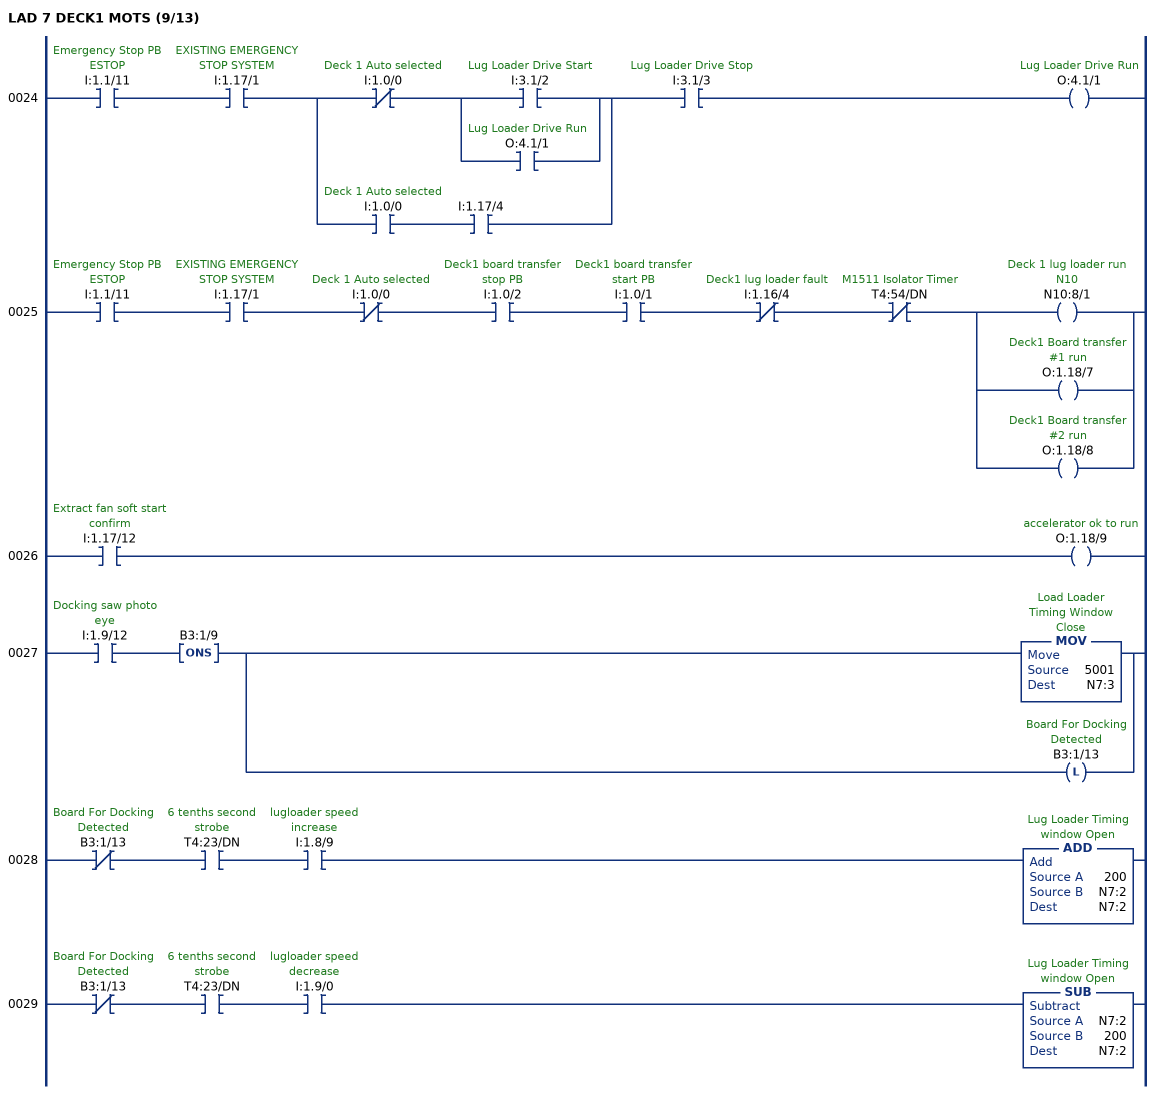
% Rung: 24 %
SOR XIC I:1.1/11 XIC I:1.17/1 BST XIO I:1.0/0 BST XIC I:3.1/2 NXB XIC O:4.1/1 BND NXB XIC I:1.0/0 XIC I:1.17/4 BND XIC I:3.1/3 OTE O:4.1/1 EOR
%   I:1.1/11  ESTOP  "Emergency Stop PB" %
%   I:1.17/1  "EXISTING EMERGENCY STOP SYSTEM" %
%   I:1.0/0  "Deck 1 Auto selected" %
%   I:3.1/2  "Lug Loader Drive Start" %
%   O:4.1/1  "Lug Loader Drive Run" %
%   I:3.1/3  "Lug Loader Drive Stop" %
% Rung: 25 %
SOR XIC I:1.1/11 XIC I:1.17/1 XIO I:1.0/0 XIC I:1.0/2 XIC I:1.0/1 XIO I:1.16/4 XIO T4:54/DN BST OTE N10:8/1 NXB OTE O:1.18/7 NXB OTE O:1.18/8 BND EOR
%   I:1.1/11  ESTOP  "Emergency Stop PB" %
%   I:1.17/1  "EXISTING EMERGENCY STOP SYSTEM" %
%   I:1.0/0  "Deck 1 Auto selected" %
%   I:1.0/2  "Deck1 board transfer stop PB" %
%   I:1.0/1  "Deck1 board transfer start PB" %
%   I:1.16/4  "Deck1 lug loader fault" %
%   T4:54  "M1511 Isolator Timer" %
%   N10:8/1  N10  "Deck 1 lug loader run" %
%   O:1.18/7  "Deck1 Board transfer #1 run" %
%   O:1.18/8  "Deck1 Board transfer #2 run" %
% Rung: 26 %
SOR XIC I:1.17/12 OTE O:1.18/9 EOR
%   I:1.17/12  "Extract fan soft start confirm" %
%   O:1.18/9  "accelerator ok to run" %
% Rung: 27 %
SOR XIC I:1.9/12 OSR B3:1/9 BST MOV 5001 N7:3 NXB OTL B3:1/13 BND EOR
%   I:1.9/12  "Docking saw photo eye" %
%   N7:3  "Load Loader Timing Window Close" %
%   B3:1/13  "Board For Docking Detected" %
% Rung: 28 %
SOR XIO B3:1/13 XIC T4:23/DN XIC I:1.8/9 ADD 200 N7:2 N7:2 EOR
%   B3:1/13  "Board For Docking Detected" %
%   T4:23/DN  "6 tenths second strobe" %
%   I:1.8/9  "lugloader speed increase" %
%   N7:2  "Lug Loader Timing window Open" %
% Rung: 29 %
SOR XIO B3:1/13 XIC T4:23/DN XIC I:1.9/0 SUB N7:2 200 N7:2 EOR
%   B3:1/13  "Board For Docking Detected" %
%   T4:23/DN  "6 tenths second strobe" %
%   I:1.9/0  "lugloader speed decrease" %
%   N7:2  "Lug Loader Timing window Open" %

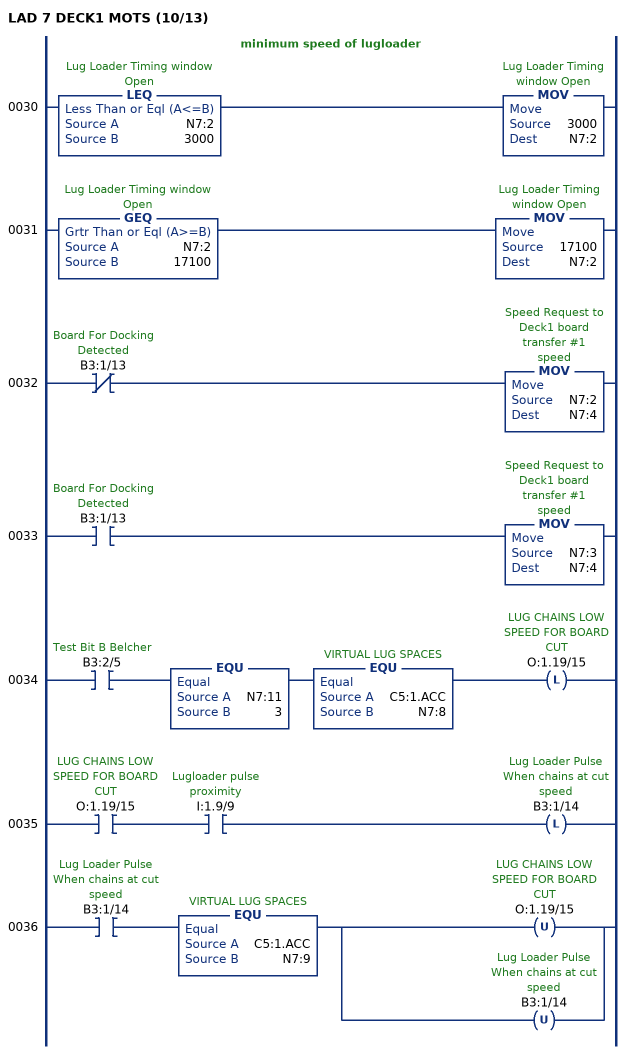
% Rung: 30 %
% TITLE: minimum speed of lugloader %
SOR LEQ N7:2 3000 MOV 3000 N7:2 EOR
%   N7:2  "Lug Loader Timing window Open" %
% Rung: 31 %
SOR GEQ N7:2 17100 MOV 17100 N7:2 EOR
%   N7:2  "Lug Loader Timing window Open" %
% Rung: 32 %
SOR XIO B3:1/13 MOV N7:2 N7:4 EOR
%   B3:1/13  "Board For Docking Detected" %
%   N7:2  "Lug Loader Timing window Open" %
%   N7:4  "Speed Request to Deck1 board transfer #1 speed" %
% Rung: 33 %
SOR XIC B3:1/13 MOV N7:3 N7:4 EOR
%   B3:1/13  "Board For Docking Detected" %
%   N7:3  "Load Loader Timing Window Close" %
%   N7:4  "Speed Request to Deck1 board transfer #1 speed" %
% Rung: 34 %
SOR XIC B3:2/5 EQU N7:11 3 EQU C5:1.ACC N7:8 OTL O:1.19/15 EOR
%   B3:2/5  "Test Bit B Belcher" %
%   C5:1  "VIRTUAL LUG SPACES" %
%   N7:8  "CUT BOARD SLOW DOWN ON" %
%   O:1.19/15  "LUG CHAINS LOW SPEED FOR BOARD CUT" %
% Rung: 35 %
SOR XIC O:1.19/15 XIC I:1.9/9 OTL B3:1/14 EOR
%   O:1.19/15  "LUG CHAINS LOW SPEED FOR BOARD CUT" %
%   I:1.9/9  "Lugloader pulse proximity" %
%   B3:1/14  "Lug Loader Pulse When chains at cut speed" %
% Rung: 36 %
SOR XIC B3:1/14 EQU C5:1.ACC N7:9 BST OTU O:1.19/15 NXB OTU B3:1/14 BND EOR
%   B3:1/14  "Lug Loader Pulse When chains at cut speed" %
%   C5:1  "VIRTUAL LUG SPACES" %
%   O:1.19/15  "LUG CHAINS LOW SPEED FOR BOARD CUT" %

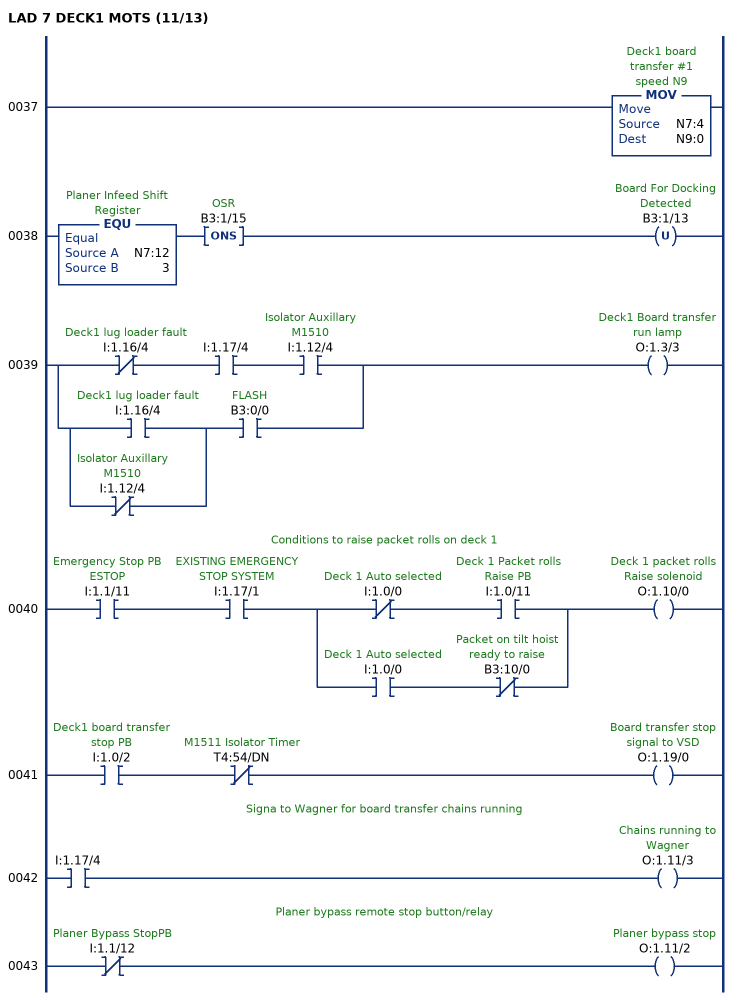
% Rung: 37 %
SOR MOV N7:4 N9:0 EOR
%   N7:4  "Speed Request to Deck1 board transfer #1 speed" %
%   N9:0  N9  "Deck1 board transfer #1 speed" %
% Rung: 38 %
SOR EQU N7:12 3 OSR B3:1/15 OTU B3:1/13 EOR
%   N7:12  "Planer Infeed Shift Register" %
%   B3:1/15  "OSR" %
%   B3:1/13  "Board For Docking Detected" %
% Rung: 39 %
SOR BST XIO I:1.16/4 XIC I:1.17/4 XIC I:1.12/4 NXB BST XIC I:1.16/4 NXB XIO I:1.12/4 BND XIC B3:0/0 BND OTE O:1.3/3 EOR
%   I:1.16/4  "Deck1 lug loader fault" %
%   I:1.12/4  "Isolator Auxillary M1510" %
%   B3:0/0  FLASH %
%   O:1.3/3  "Deck1 Board transfer run lamp" %
% Rung: 40 %
% Conditions to raise packet rolls on deck 1 %
SOR XIC I:1.1/11 XIC I:1.17/1 BST XIO I:1.0/0 XIC I:1.0/11 NXB XIC I:1.0/0 XIO B3:10/0 BND OTE O:1.10/0 EOR
%   I:1.1/11  ESTOP  "Emergency Stop PB" %
%   I:1.17/1  "EXISTING EMERGENCY STOP SYSTEM" %
%   I:1.0/0  "Deck 1 Auto selected" %
%   I:1.0/11  "Deck 1 Packet rolls Raise PB" %
%   B3:10/0  "Packet on tilt hoist ready to raise" %
%   O:1.10/0  "Deck 1 packet rolls Raise solenoid" %
% Rung: 41 %
SOR XIC I:1.0/2 XIO T4:54/DN OTE O:1.19/0 EOR
%   I:1.0/2  "Deck1 board transfer stop PB" %
%   T4:54  "M1511 Isolator Timer" %
%   O:1.19/0  "Board transfer stop signal to VSD" %
% Rung: 42 %
% Signa to Wagner for board transfer chains running %
SOR XIC I:1.17/4 OTE O:1.11/3 EOR
%   O:1.11/3  "Chains running to Wagner" %
% Rung: 43 %
% Planer bypass remote stop button/relay %
SOR XIO I:1.1/12 OTE O:1.11/2 EOR
%   I:1.1/12  "Planer Bypass StopPB" %
%   O:1.11/2  "Planer bypass stop" %

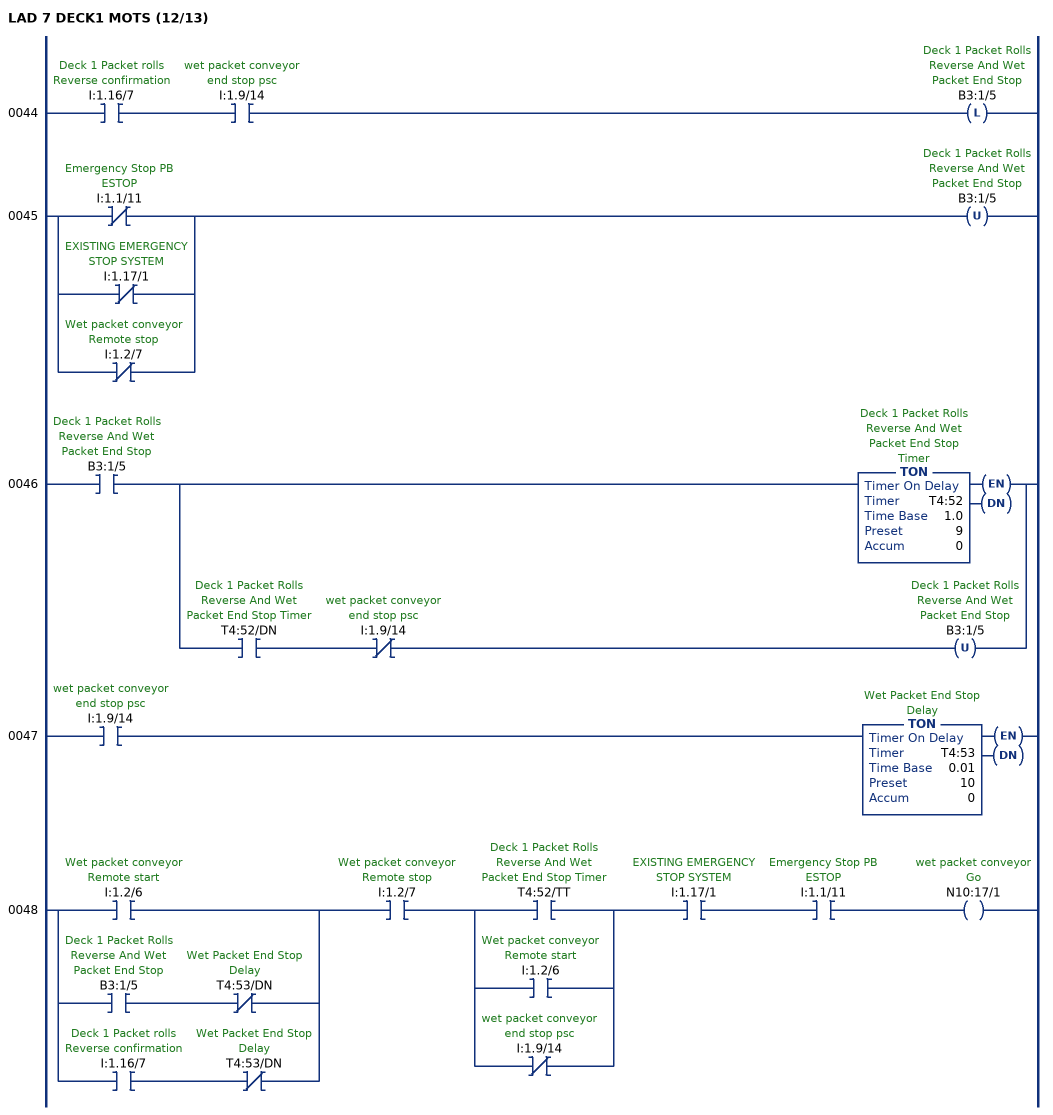
% Rung: 44 %
SOR XIC I:1.16/7 XIC I:1.9/14 OTL B3:1/5 EOR
%   I:1.16/7  "Deck 1 Packet rolls Reverse confirmation" %
%   I:1.9/14  "wet packet conveyor end stop psc" %
%   B3:1/5  "Deck 1 Packet Rolls Reverse And Wet Packet End Stop" %
% Rung: 45 %
SOR BST XIO I:1.1/11 NXB XIO I:1.17/1 NXB XIO I:1.2/7 BND OTU B3:1/5 EOR
%   I:1.1/11  ESTOP  "Emergency Stop PB" %
%   I:1.17/1  "EXISTING EMERGENCY STOP SYSTEM" %
%   I:1.2/7  "Wet packet conveyor Remote stop" %
%   B3:1/5  "Deck 1 Packet Rolls Reverse And Wet Packet End Stop" %
% Rung: 46 %
SOR XIC B3:1/5 BST TON T4:52 1.0 9 0 NXB XIC T4:52/DN XIO I:1.9/14 OTU B3:1/5 BND EOR
%   B3:1/5  "Deck 1 Packet Rolls Reverse And Wet Packet End Stop" %
%   T4:52  "Deck 1 Packet Rolls Reverse And Wet Packet End Stop Timer" %
%   I:1.9/14  "wet packet conveyor end stop psc" %
% Rung: 47 %
SOR XIC I:1.9/14 TON T4:53 0.01 10 0 EOR
%   I:1.9/14  "wet packet conveyor end stop psc" %
%   T4:53  "Wet Packet End Stop Delay" %
% Rung: 48 %
SOR BST XIC I:1.2/6 NXB XIC B3:1/5 XIO T4:53/DN NXB XIC I:1.16/7 XIO T4:53/DN BND XIC I:1.2/7 BST XIC T4:52/TT NXB XIC I:1.2/6 NXB XIO I:1.9/14 BND XIC I:1.17/1 XIC I:1.1/11 OTE N10:17/1 EOR
%   I:1.2/6  "Wet packet conveyor Remote start" %
%   B3:1/5  "Deck 1 Packet Rolls Reverse And Wet Packet End Stop" %
%   T4:53  "Wet Packet End Stop Delay" %
%   I:1.16/7  "Deck 1 Packet rolls Reverse confirmation" %
%   I:1.2/7  "Wet packet conveyor Remote stop" %
%   T4:52  "Deck 1 Packet Rolls Reverse And Wet Packet End Stop Timer" %
%   I:1.9/14  "wet packet conveyor end stop psc" %
%   I:1.17/1  "EXISTING EMERGENCY STOP SYSTEM" %
%   I:1.1/11  ESTOP  "Emergency Stop PB" %
%   N10:17/1  "wet packet conveyor Go" %

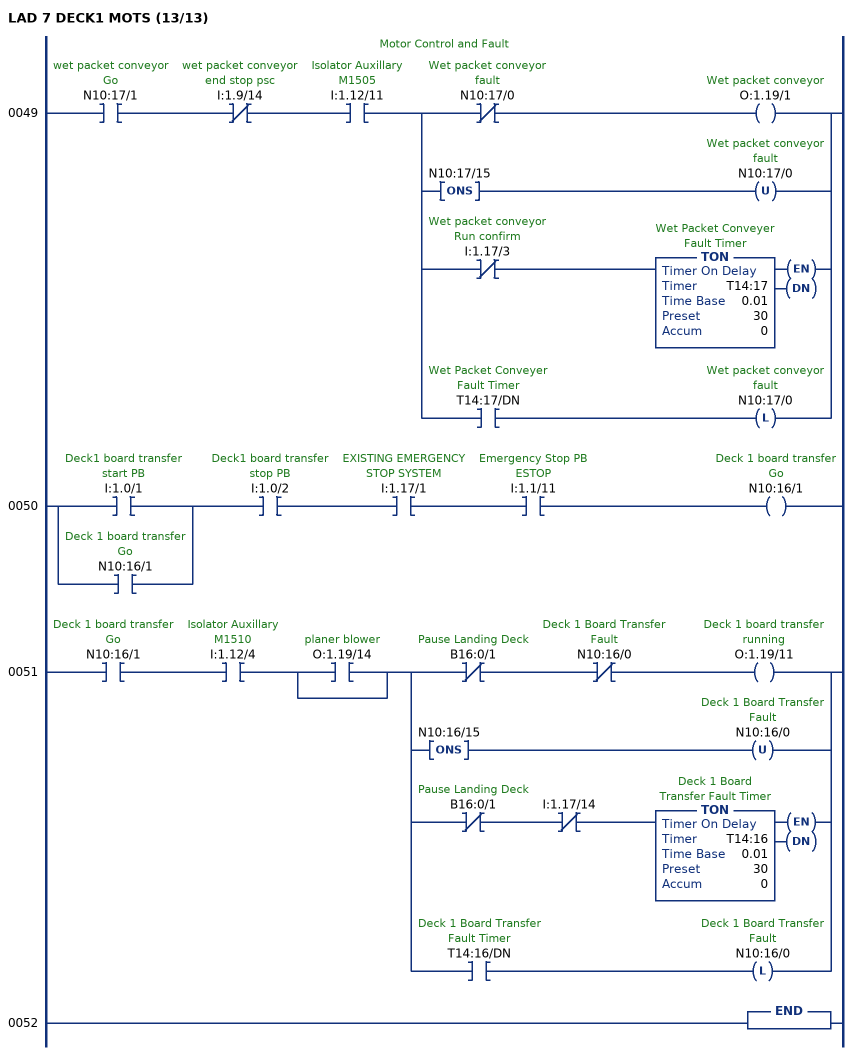
% Rung: 49 %
% Motor Control and Fault %
SOR XIC N10:17/1 XIO I:1.9/14 XIC I:1.12/11 BST XIO N10:17/0 OTE O:1.19/1 NXB OSR N10:17/15 OTU N10:17/0 NXB XIO I:1.17/3 TON T14:17 0.01 30 0 NXB XIC T14:17/DN OTL N10:17/0 BND EOR
%   N10:17/1  "wet packet conveyor Go" %
%   I:1.9/14  "wet packet conveyor end stop psc" %
%   I:1.12/11  "Isolator Auxillary M1505" %
%   N10:17/0  "Wet packet conveyor fault" %
%   O:1.19/1  "Wet packet conveyor" %
%   I:1.17/3  "Wet packet conveyor Run confirm" %
%   T14:17  "Wet Packet Conveyer Fault Timer" %
% Rung: 50 %
SOR BST XIC I:1.0/1 NXB XIC N10:16/1 BND XIC I:1.0/2 XIC I:1.17/1 XIC I:1.1/11 OTE N10:16/1 EOR
%   I:1.0/1  "Deck1 board transfer start PB" %
%   N10:16/1  "Deck 1 board transfer Go" %
%   I:1.0/2  "Deck1 board transfer stop PB" %
%   I:1.17/1  "EXISTING EMERGENCY STOP SYSTEM" %
%   I:1.1/11  ESTOP  "Emergency Stop PB" %
% Rung: 51 %
SOR XIC N10:16/1 XIC I:1.12/4 BST XIC O:1.19/14 NXB BND BST XIO B16:0/1 XIO N10:16/0 OTE O:1.19/11 NXB OSR N10:16/15 OTU N10:16/0 NXB XIO B16:0/1 XIO I:1.17/14 TON T14:16 0.01 30 0 NXB XIC T14:16/DN OTL N10:16/0 BND EOR
%   N10:16/1  "Deck 1 board transfer Go" %
%   I:1.12/4  "Isolator Auxillary M1510" %
%   O:1.19/14  "planer blower" %
%   B16:0/1  "Pause Landing Deck" %
%   N10:16/0  "Deck 1 Board Transfer Fault" %
%   O:1.19/11  "Deck 1 board transfer running" %
%   T14:16  "Deck 1 Board Transfer Fault Timer" %
% Rung: 52 %
SOR END EOR

LADDER 8 "EXTRACTFAN"
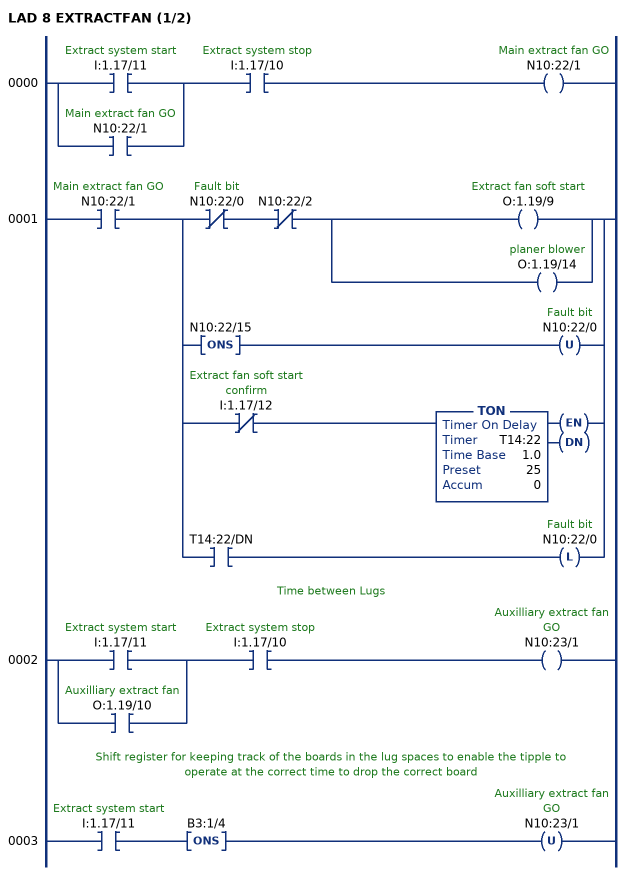
% Rung: 0 %
SOR BST XIC I:1.17/11 NXB XIC N10:22/1 BND XIC I:1.17/10 OTE N10:22/1 EOR
%   I:1.17/11  "Extract system start" %
%   N10:22/1  "Main extract fan GO" %
%   I:1.17/10  "Extract system stop" %
% Rung: 1 %
SOR XIC N10:22/1 BST XIO N10:22/0 XIO N10:22/2 BST OTE O:1.19/9 NXB OTE O:1.19/14 BND NXB OSR N10:22/15 OTU N10:22/0 NXB XIO I:1.17/12 TON T14:22 1.0 25 0 NXB XIC T14:22/DN OTL N10:22/0 BND EOR
%   N10:22/1  "Main extract fan GO" %
%   N10:22/0  "Fault bit" %
%   O:1.19/9  "Extract fan soft start" %
%   O:1.19/14  "planer blower" %
%   I:1.17/12  "Extract fan soft start confirm" %
% Rung: 2 %
% Time between Lugs %
SOR BST XIC I:1.17/11 NXB XIC O:1.19/10 BND XIC I:1.17/10 OTE N10:23/1 EOR
%   I:1.17/11  "Extract system start" %
%   O:1.19/10  "Auxilliary extract fan" %
%   I:1.17/10  "Extract system stop" %
%   N10:23/1  "Auxilliary extract fan GO" %
% Rung: 3 %
% Shift register for keeping track of the boards in the lug spaces to enable the tipple to operate at the correct time to drop the correct board %
SOR XIC I:1.17/11 OSR B3:1/4 OTU N10:23/1 EOR
%   I:1.17/11  "Extract system start" %
%   N10:23/1  "Auxilliary extract fan GO" %

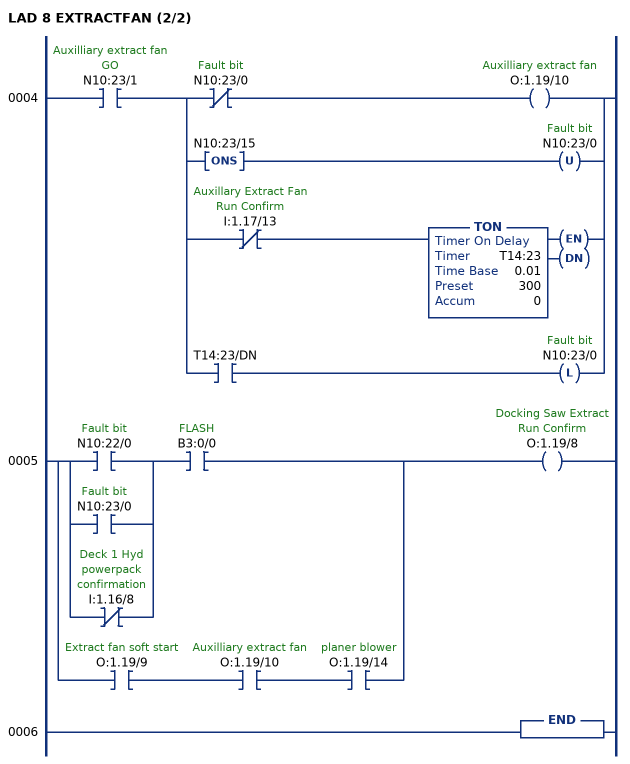
% Rung: 4 %
SOR XIC N10:23/1 BST XIO N10:23/0 OTE O:1.19/10 NXB OSR N10:23/15 OTU N10:23/0 NXB XIO I:1.17/13 TON T14:23 0.01 300 0 NXB XIC T14:23/DN OTL N10:23/0 BND EOR
%   N10:23/1  "Auxilliary extract fan GO" %
%   N10:23/0  "Fault bit" %
%   O:1.19/10  "Auxilliary extract fan" %
%   I:1.17/13  "Auxillary Extract Fan Run Confirm" %
% Rung: 5 %
SOR BST BST XIC N10:22/0 NXB BST XIC N10:23/0 NXB XIO I:1.16/8 BND BND XIC B3:0/0 NXB XIC O:1.19/9 XIC O:1.19/10 XIC O:1.19/14 BND OTE O:1.19/8 EOR
%   N10:22/0  "Fault bit" %
%   N10:23/0  "Fault bit" %
%   I:1.16/8  "Deck 1 Hyd powerpack confirmation" %
%   B3:0/0  FLASH %
%   O:1.19/9  "Extract fan soft start" %
%   O:1.19/10  "Auxilliary extract fan" %
%   O:1.19/14  "planer blower" %
%   O:1.19/8  "Docking Saw Extract Run Confirm" %
% Rung: 6 %
SOR END EOR

LADDER 9 "BLOCKTX"
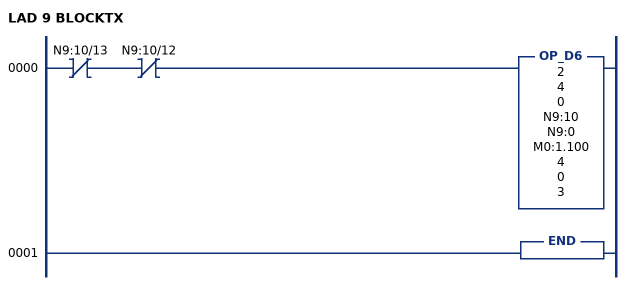
% Rung: 0 %
SOR XIO N9:10/13 XIO N9:10/12 OP_D6 2 4 0 N9:10 N9:0 M0:1.100 4 0 3 EOR
%   N9:10  BTW_CTRL  "Remote IO Analog Block Transfer Control" %
%   N9:0  N9  "Deck1 board transfer #1 speed" %
% Rung: 1 %
SOR END EOR

LADDER 14 "DECK2 MOTS"
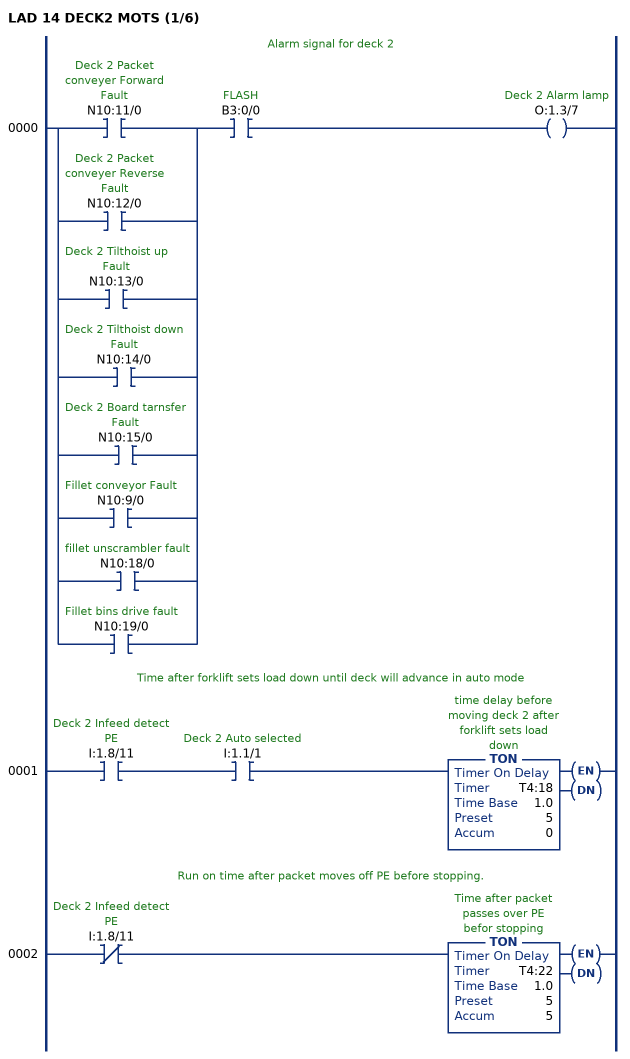
% Rung: 0 %
% Alarm signal for deck 2 %
SOR BST XIC N10:11/0 NXB XIC N10:12/0 NXB XIC N10:13/0 NXB XIC N10:14/0 NXB XIC N10:15/0 NXB XIC N10:9/0 NXB XIC N10:18/0 NXB XIC N10:19/0 BND XIC B3:0/0 OTE O:1.3/7 EOR
%   N10:11/0  "Deck 2 Packet conveyer Forward Fault" %
%   N10:12/0  "Deck 2 Packet conveyer Reverse Fault" %
%   N10:13/0  "Deck 2 Tilthoist up Fault" %
%   N10:14/0  "Deck 2 Tilthoist down Fault" %
%   N10:15/0  "Deck 2 Board tarnsfer Fault" %
%   N10:9/0  "Fillet conveyor Fault" %
%   N10:18/0  "fillet unscrambler fault" %
%   N10:19/0  "Fillet bins drive fault" %
%   B3:0/0  FLASH %
%   O:1.3/7  "Deck 2 Alarm lamp" %
% Rung: 1 %
% Time after forklift sets load down until deck will advance in auto mode %
SOR XIC I:1.8/11 XIC I:1.1/1 TON T4:18 1.0 5 0 EOR
%   I:1.8/11  "Deck 2 Infeed detect PE" %
%   I:1.1/1  "Deck 2 Auto selected" %
%   T4:18  "time delay before moving deck 2 after forklift sets load down" %
% Rung: 2 %
% Run on time after packet moves off PE before stopping. %
SOR XIO I:1.8/11 TON T4:22 1.0 5 5 EOR
%   I:1.8/11  "Deck 2 Infeed detect PE" %
%   T4:22  "Time after packet passes over PE befor stopping" %

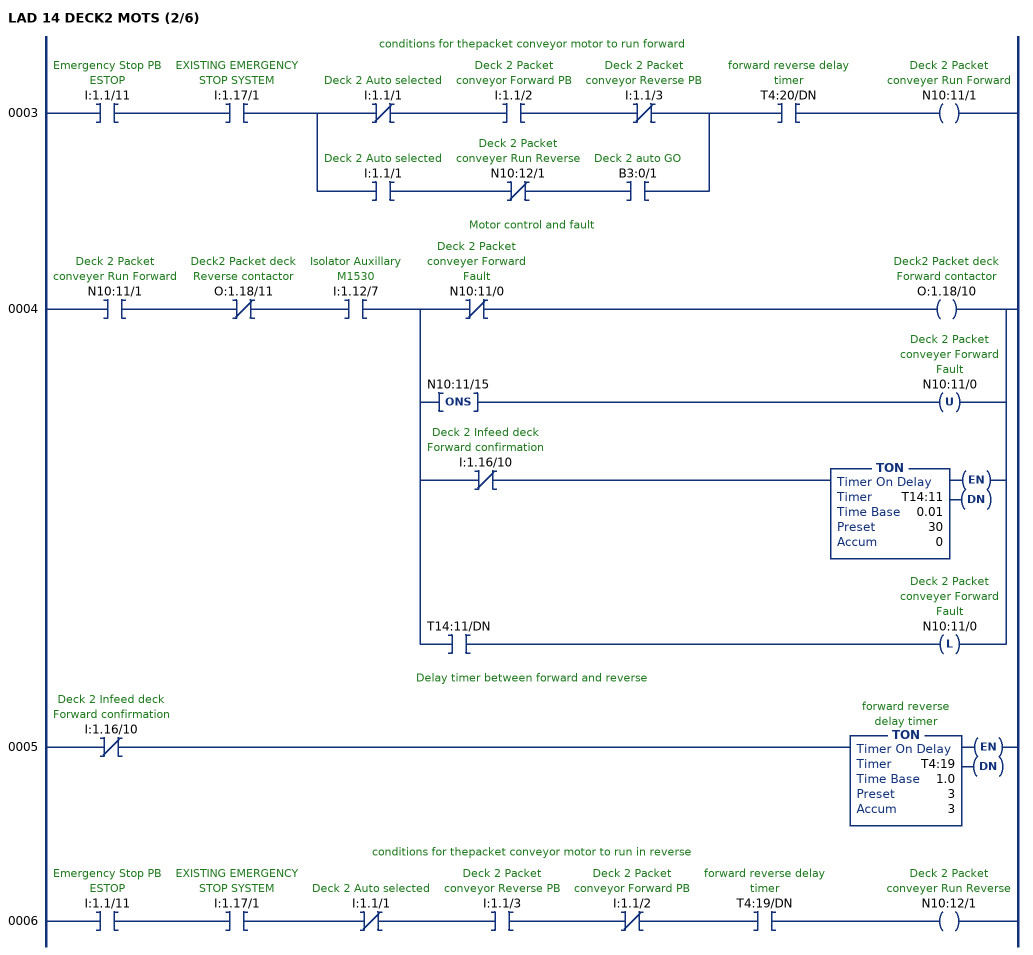
% Rung: 3 %
% conditions for thepacket conveyor motor to run forward %
SOR XIC I:1.1/11 XIC I:1.17/1 BST XIO I:1.1/1 XIC I:1.1/2 XIO I:1.1/3 NXB XIC I:1.1/1 XIO N10:12/1 XIC B3:0/1 BND XIC T4:20/DN OTE N10:11/1 EOR
%   I:1.1/11  ESTOP  "Emergency Stop PB" %
%   I:1.17/1  "EXISTING EMERGENCY STOP SYSTEM" %
%   I:1.1/1  "Deck 2 Auto selected" %
%   I:1.1/2  "Deck 2 Packet conveyor Forward PB" %
%   I:1.1/3  "Deck 2 Packet conveyor Reverse PB" %
%   N10:12/1  "Deck 2 Packet conveyer Run Reverse" %
%   B3:0/1  "Deck 2 auto GO" %
%   T4:20  "forward reverse delay timer" %
%   N10:11/1  "Deck 2 Packet conveyer Run Forward" %
% Rung: 4 %
% Motor control and fault %
SOR XIC N10:11/1 XIO O:1.18/11 XIC I:1.12/7 BST XIO N10:11/0 OTE O:1.18/10 NXB OSR N10:11/15 OTU N10:11/0 NXB XIO I:1.16/10 TON T14:11 0.01 30 0 NXB XIC T14:11/DN OTL N10:11/0 BND EOR
%   N10:11/1  "Deck 2 Packet conveyer Run Forward" %
%   O:1.18/11  "Deck2 Packet deck Reverse contactor" %
%   I:1.12/7  "Isolator Auxillary M1530" %
%   N10:11/0  "Deck 2 Packet conveyer Forward Fault" %
%   O:1.18/10  "Deck2 Packet deck Forward contactor" %
%   I:1.16/10  "Deck 2 Infeed deck Forward confirmation" %
% Rung: 5 %
% Delay timer between forward and reverse %
SOR XIO I:1.16/10 TON T4:19 1.0 3 3 EOR
%   I:1.16/10  "Deck 2 Infeed deck Forward confirmation" %
%   T4:19  "forward reverse delay timer" %
% Rung: 6 %
% conditions for thepacket conveyor motor to run in reverse %
SOR XIC I:1.1/11 XIC I:1.17/1 XIO I:1.1/1 XIC I:1.1/3 XIO I:1.1/2 XIC T4:19/DN OTE N10:12/1 EOR
%   I:1.1/11  ESTOP  "Emergency Stop PB" %
%   I:1.17/1  "EXISTING EMERGENCY STOP SYSTEM" %
%   I:1.1/1  "Deck 2 Auto selected" %
%   I:1.1/3  "Deck 2 Packet conveyor Reverse PB" %
%   I:1.1/2  "Deck 2 Packet conveyor Forward PB" %
%   T4:19  "forward reverse delay timer" %
%   N10:12/1  "Deck 2 Packet conveyer Run Reverse" %

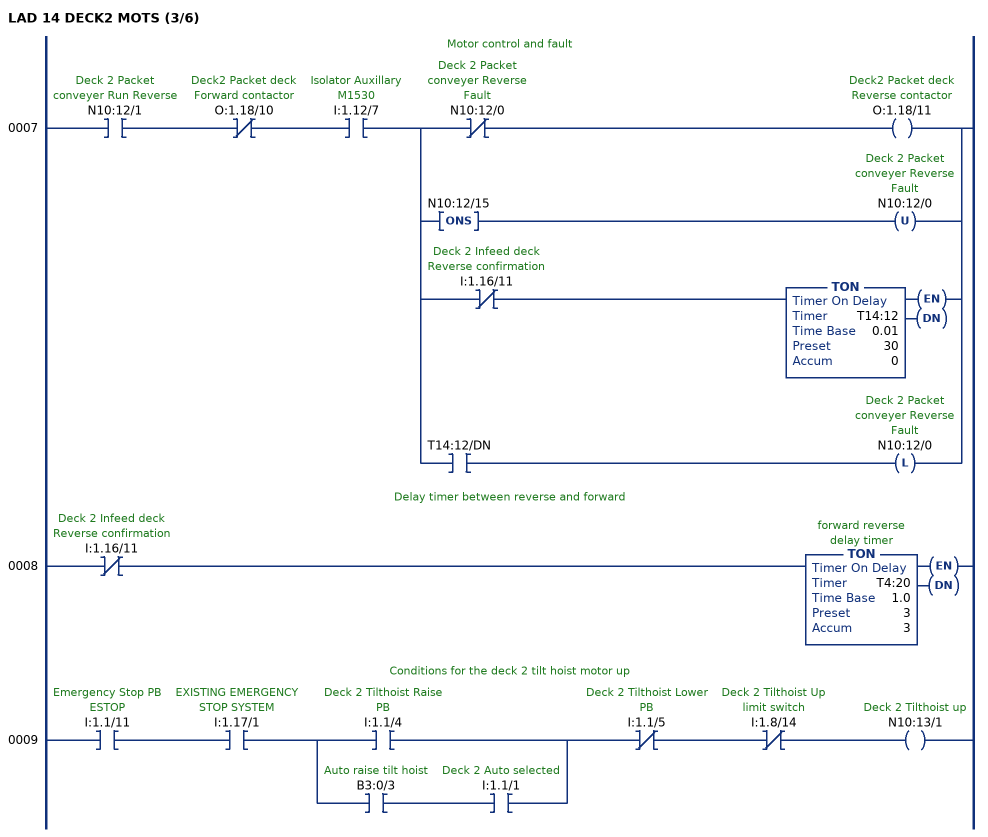
% Rung: 7 %
% Motor control and fault %
SOR XIC N10:12/1 XIO O:1.18/10 XIC I:1.12/7 BST XIO N10:12/0 OTE O:1.18/11 NXB OSR N10:12/15 OTU N10:12/0 NXB XIO I:1.16/11 TON T14:12 0.01 30 0 NXB XIC T14:12/DN OTL N10:12/0 BND EOR
%   N10:12/1  "Deck 2 Packet conveyer Run Reverse" %
%   O:1.18/10  "Deck2 Packet deck Forward contactor" %
%   I:1.12/7  "Isolator Auxillary M1530" %
%   N10:12/0  "Deck 2 Packet conveyer Reverse Fault" %
%   O:1.18/11  "Deck2 Packet deck Reverse contactor" %
%   I:1.16/11  "Deck 2 Infeed deck Reverse confirmation" %
% Rung: 8 %
% Delay timer between reverse and forward %
SOR XIO I:1.16/11 TON T4:20 1.0 3 3 EOR
%   I:1.16/11  "Deck 2 Infeed deck Reverse confirmation" %
%   T4:20  "forward reverse delay timer" %
% Rung: 9 %
% Conditions for the deck 2 tilt hoist motor up %
SOR XIC I:1.1/11 XIC I:1.17/1 BST XIC I:1.1/4 NXB XIC B3:0/3 XIC I:1.1/1 BND XIO I:1.1/5 XIO I:1.8/14 OTE N10:13/1 EOR
%   I:1.1/11  ESTOP  "Emergency Stop PB" %
%   I:1.17/1  "EXISTING EMERGENCY STOP SYSTEM" %
%   I:1.1/4  "Deck 2 Tilthoist Raise PB" %
%   B3:0/3  "Auto raise tilt hoist" %
%   I:1.1/1  "Deck 2 Auto selected" %
%   I:1.1/5  "Deck 2 Tilthoist Lower PB" %
%   I:1.8/14  "Deck 2 Tilthoist Up limit switch" %
%   N10:13/1  "Deck 2 Tilthoist up" %

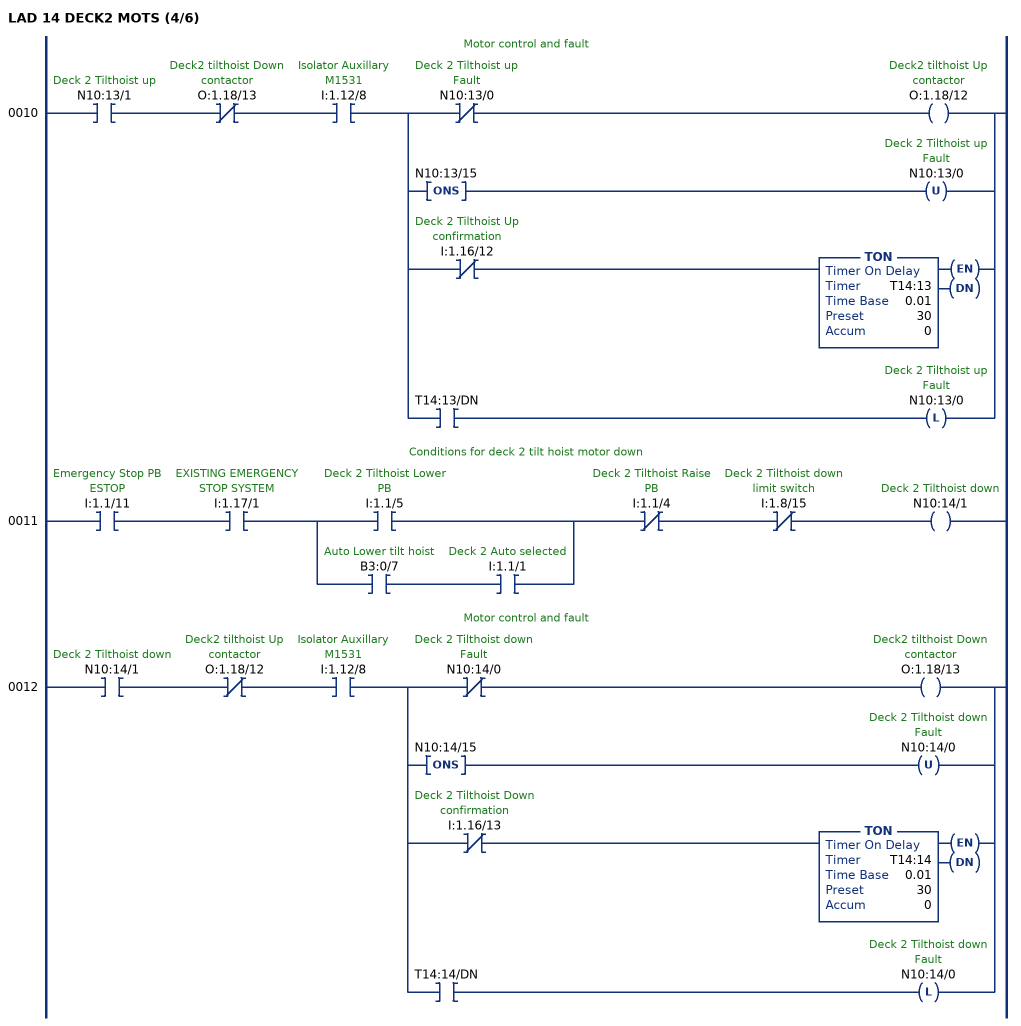
% Rung: 10 %
% Motor control and fault %
SOR XIC N10:13/1 XIO O:1.18/13 XIC I:1.12/8 BST XIO N10:13/0 OTE O:1.18/12 NXB OSR N10:13/15 OTU N10:13/0 NXB XIO I:1.16/12 TON T14:13 0.01 30 0 NXB XIC T14:13/DN OTL N10:13/0 BND EOR
%   N10:13/1  "Deck 2 Tilthoist up" %
%   O:1.18/13  "Deck2 tilthoist Down contactor" %
%   I:1.12/8  "Isolator Auxillary M1531" %
%   N10:13/0  "Deck 2 Tilthoist up Fault" %
%   O:1.18/12  "Deck2 tilthoist Up contactor" %
%   I:1.16/12  "Deck 2 Tilthoist Up confirmation" %
% Rung: 11 %
% Conditions for deck 2 tilt hoist motor down %
SOR XIC I:1.1/11 XIC I:1.17/1 BST XIC I:1.1/5 NXB XIC B3:0/7 XIC I:1.1/1 BND XIO I:1.1/4 XIO I:1.8/15 OTE N10:14/1 EOR
%   I:1.1/11  ESTOP  "Emergency Stop PB" %
%   I:1.17/1  "EXISTING EMERGENCY STOP SYSTEM" %
%   I:1.1/5  "Deck 2 Tilthoist Lower PB" %
%   B3:0/7  "Auto Lower tilt hoist" %
%   I:1.1/1  "Deck 2 Auto selected" %
%   I:1.1/4  "Deck 2 Tilthoist Raise PB" %
%   I:1.8/15  "Deck 2 Tilthoist down limit switch" %
%   N10:14/1  "Deck 2 Tilthoist down" %
% Rung: 12 %
% Motor control and fault %
SOR XIC N10:14/1 XIO O:1.18/12 XIC I:1.12/8 BST XIO N10:14/0 OTE O:1.18/13 NXB OSR N10:14/15 OTU N10:14/0 NXB XIO I:1.16/13 TON T14:14 0.01 30 0 NXB XIC T14:14/DN OTL N10:14/0 BND EOR
%   N10:14/1  "Deck 2 Tilthoist down" %
%   O:1.18/12  "Deck2 tilthoist Up contactor" %
%   I:1.12/8  "Isolator Auxillary M1531" %
%   N10:14/0  "Deck 2 Tilthoist down Fault" %
%   O:1.18/13  "Deck2 tilthoist Down contactor" %
%   I:1.16/13  "Deck 2 Tilthoist Down confirmation" %

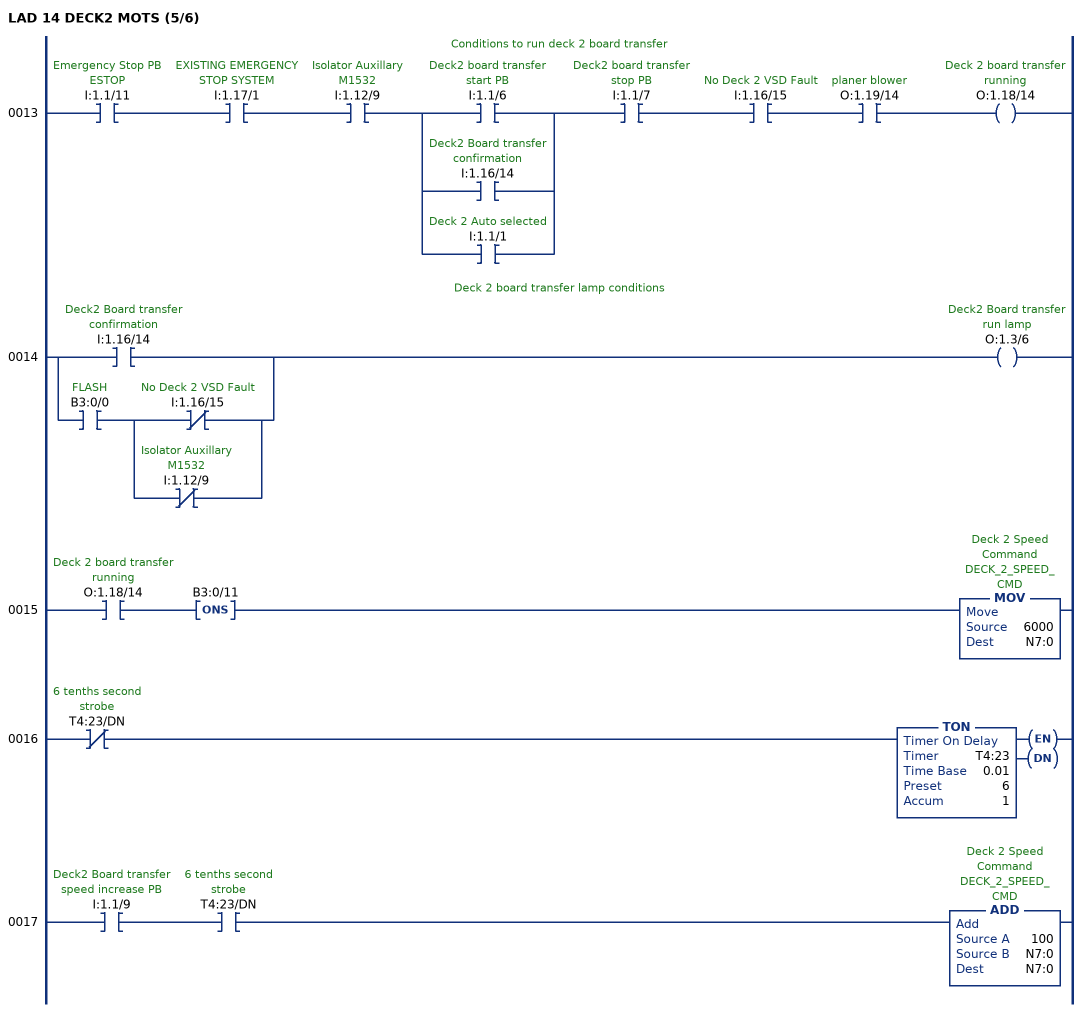
% Rung: 13 %
% Conditions to run deck 2 board transfer %
SOR XIC I:1.1/11 XIC I:1.17/1 XIC I:1.12/9 BST XIC I:1.1/6 NXB BST XIC I:1.16/14 NXB XIC I:1.1/1 BND BND XIC I:1.1/7 XIC I:1.16/15 XIC O:1.19/14 OTE O:1.18/14 EOR
%   I:1.1/11  ESTOP  "Emergency Stop PB" %
%   I:1.17/1  "EXISTING EMERGENCY STOP SYSTEM" %
%   I:1.12/9  "Isolator Auxillary M1532" %
%   I:1.1/6  "Deck2 board transfer start PB" %
%   I:1.16/14  "Deck2 Board transfer confirmation" %
%   I:1.1/1  "Deck 2 Auto selected" %
%   I:1.1/7  "Deck2 board transfer stop PB" %
%   I:1.16/15  "No Deck 2 VSD Fault" %
%   O:1.19/14  "planer blower" %
%   O:1.18/14  "Deck 2 board transfer running" %
% Rung: 14 %
% Deck 2 board transfer lamp conditions %
SOR BST XIC I:1.16/14 NXB XIC B3:0/0 BST XIO I:1.16/15 NXB XIO I:1.12/9 BND BND OTE O:1.3/6 EOR
%   I:1.16/14  "Deck2 Board transfer confirmation" %
%   B3:0/0  FLASH %
%   I:1.16/15  "No Deck 2 VSD Fault" %
%   I:1.12/9  "Isolator Auxillary M1532" %
%   O:1.3/6  "Deck2 Board transfer run lamp" %
% Rung: 15 %
SOR XIC O:1.18/14 OSR B3:0/11 MOV 6000 N7:0 EOR
%   O:1.18/14  "Deck 2 board transfer running" %
%   N7:0  DECK_2_SPEED_CMD  "Deck 2 Speed Command" %
% Rung: 16 %
SOR XIO T4:23/DN TON T4:23 0.01 6 1 EOR
%   T4:23/DN  "6 tenths second strobe" %
% Rung: 17 %
SOR XIC I:1.1/9 XIC T4:23/DN ADD 100 N7:0 N7:0 EOR
%   I:1.1/9  "Deck2 Board transfer speed increase PB" %
%   T4:23/DN  "6 tenths second strobe" %
%   N7:0  DECK_2_SPEED_CMD  "Deck 2 Speed Command" %

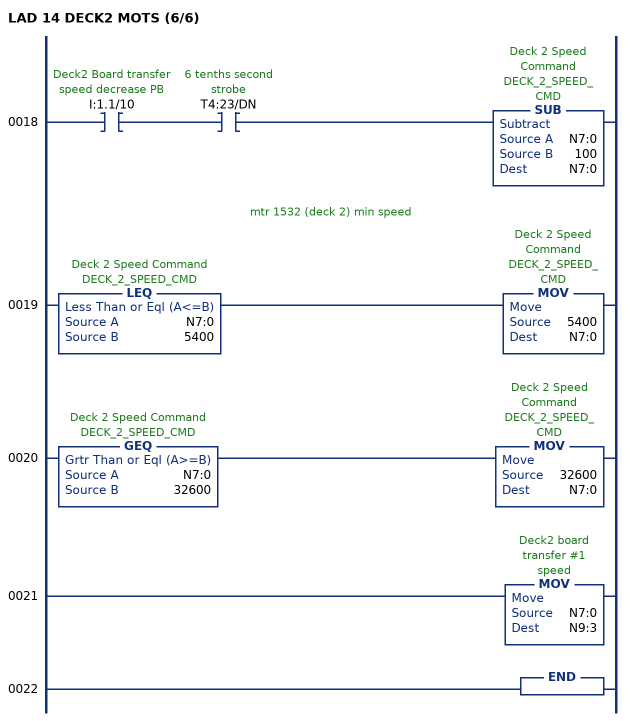
% Rung: 18 %
SOR XIC I:1.1/10 XIC T4:23/DN SUB N7:0 100 N7:0 EOR
%   I:1.1/10  "Deck2 Board transfer speed decrease PB" %
%   T4:23/DN  "6 tenths second strobe" %
%   N7:0  DECK_2_SPEED_CMD  "Deck 2 Speed Command" %
% Rung: 19 %
% mtr 1532 (deck 2) min speed %
SOR LEQ N7:0 5400 MOV 5400 N7:0 EOR
%   N7:0  DECK_2_SPEED_CMD  "Deck 2 Speed Command" %
% Rung: 20 %
SOR GEQ N7:0 32600 MOV 32600 N7:0 EOR
%   N7:0  DECK_2_SPEED_CMD  "Deck 2 Speed Command" %
% Rung: 21 %
SOR MOV N7:0 N9:3 EOR
%   N7:0  DECK_2_SPEED_CMD  "Deck 2 Speed Command" %
%   N9:3  "Deck2 board transfer #1 speed" %
% Rung: 22 %
SOR END EOR

LADDER 15 "ENCODER"
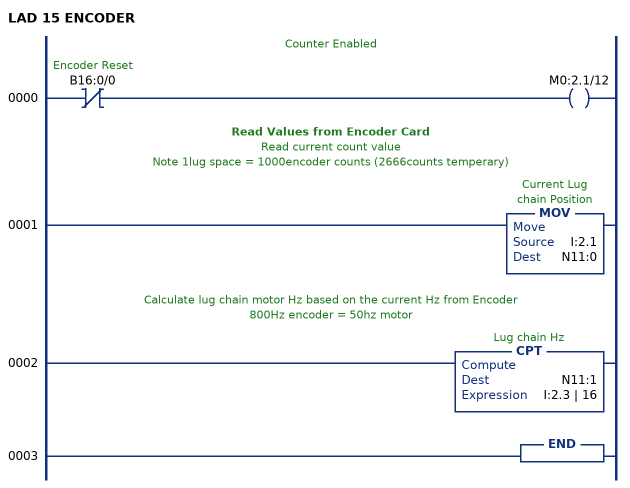
% Rung: 0 %
% Counter Enabled %
SOR XIO B16:0/0 OTE M0:2.1/12 EOR
%   B16:0/0  "Encoder Reset" %
% Rung: 1 %
% TITLE: Read Values from Encoder Card %
% Read current count value
% Note 1lug space = 1000encoder counts (2666counts temperary) %
SOR MOV I:2.1 N11:0 EOR
%   I:2.1  "Current Encoder Counts" %
%   N11:0  "Current Lug chain Position" %
% Rung: 2 %
% Calculate lug chain motor Hz based on the current Hz from Encoder
% 800Hz encoder = 50hz motor %
SOR CPT N11:1 " I:2.3 | 16 " EOR
%   N11:1  "Lug chain Hz" %
%   I:2.3  "Counter rate in Hz" %
% Rung: 3 %
SOR END EOR

LADDER 16 "FEED_CONTR"
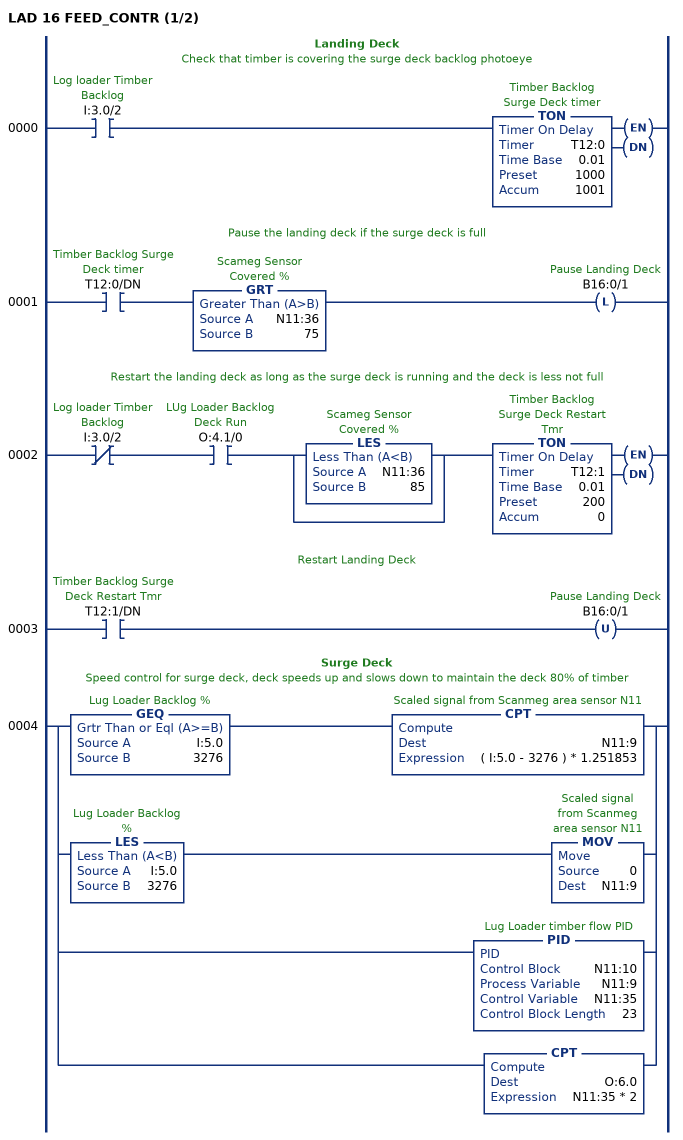
% Rung: 0 %
% TITLE: Landing Deck %
% Check that timber is covering the surge deck backlog photoeye %
SOR XIC I:3.0/2 TON T12:0 0.01 1000 1001 EOR
%   I:3.0/2  "Log loader Timber Backlog" %
%   T12:0  "Timber Backlog Surge Deck timer" %
% Rung: 1 %
% Pause the landing deck if the surge deck is full %
SOR XIC T12:0/DN GRT N11:36 75 OTL B16:0/1 EOR
%   T12:0  "Timber Backlog Surge Deck timer" %
%   N11:36  "Scameg Sensor Covered %" %
%   B16:0/1  "Pause Landing Deck" %
% Rung: 2 %
% Restart the landing deck as long as the surge deck is running and the deck is less not full %
SOR XIO I:3.0/2 XIC O:4.1/0 BST LES N11:36 85 NXB BND TON T12:1 0.01 200 0 EOR
%   I:3.0/2  "Log loader Timber Backlog" %
%   O:4.1/0  "LUg Loader Backlog Deck Run" %
%   N11:36  "Scameg Sensor Covered %" %
%   T12:1  "Timber Backlog Surge Deck Restart Tmr" %
% Rung: 3 %
% Restart Landing Deck %
SOR XIC T12:1/DN OTU B16:0/1 EOR
%   T12:1  "Timber Backlog Surge Deck Restart Tmr" %
%   B16:0/1  "Pause Landing Deck" %
% Rung: 4 %
% TITLE: Surge Deck %
% Speed control for surge deck, deck speeds up and slows down to maintain the deck 80% of timber %
SOR BST BST GEQ I:5.0 3276 CPT N11:9 " ( I:5.0 - 3276 ) * 1.251853 " NXB LES I:5.0 3276 MOV 0 N11:9 BND NXB PID N11:10 N11:9 N11:35 23 NXB CPT O:6.0 " N11:35 * 2 " BND EOR
%   I:5.0  "Lug Loader Backlog %" %
%   N11:9  N11  "Scaled signal from Scanmeg area sensor" %
%   N11:10  "Lug Loader timber flow PID" %

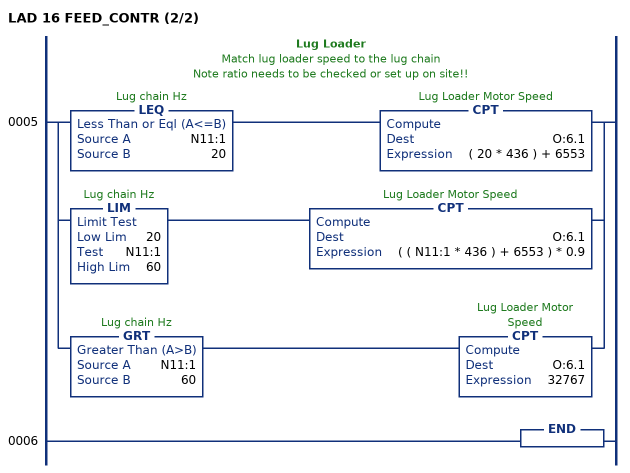
% Rung: 5 %
% TITLE: Lug Loader %
% Match lug loader speed to the lug chain
% Note ratio needs to be checked or set up on site!! %
SOR BST LEQ N11:1 20 CPT O:6.1 " ( 20 * 436 ) + 6553 " NXB LIM 20 N11:1 60 CPT O:6.1 " ( ( N11:1 * 436 ) + 6553 ) * 0.9 " NXB GRT N11:1 60 CPT O:6.1 "  32767 " BND EOR
%   N11:1  "Lug chain Hz" %
%   O:6.1  "Lug Loader Motor Speed" %
% Rung: 6 %
SOR END EOR

LADDER 17 "SCELUGLOAD"
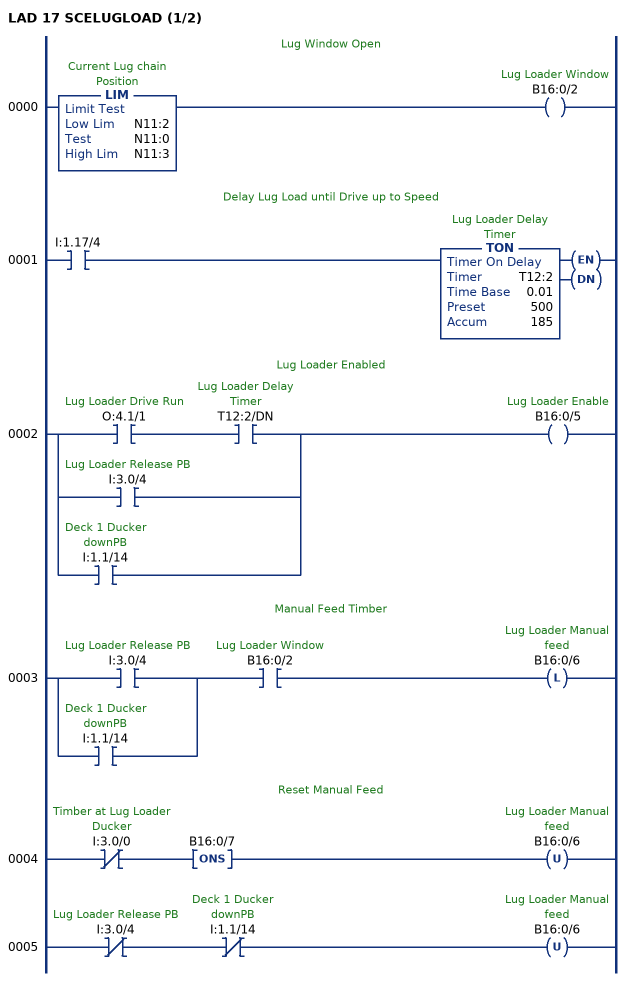
% Rung: 0 %
% Lug Window Open %
SOR LIM N11:2 N11:0 N11:3 OTE B16:0/2 EOR
%   N11:2  "Lug Loader Timing window Open" %
%   N11:0  "Current Lug chain Position" %
%   N11:3  "Load Loader Timing Window Close" %
%   B16:0/2  "Lug Loader Window" %
% Rung: 1 %
% Delay Lug Load until Drive up to Speed %
SOR XIC I:1.17/4 TON T12:2 0.01 500 185 EOR
%   T12:2  "Lug Loader Delay Timer" %
% Rung: 2 %
% Lug Loader Enabled %
SOR BST XIC O:4.1/1 XIC T12:2/DN NXB BST XIC I:3.0/4 NXB XIC I:1.1/14 BND BND OTE B16:0/5 EOR
%   O:4.1/1  "Lug Loader Drive Run" %
%   T12:2  "Lug Loader Delay Timer" %
%   I:3.0/4  "Lug Loader Release PB" %
%   I:1.1/14  "Deck 1 Ducker downPB" %
%   B16:0/5  "Lug Loader Enable" %
% Rung: 3 %
% Manual Feed Timber %
SOR BST XIC I:3.0/4 NXB XIC I:1.1/14 BND XIC B16:0/2 OTL B16:0/6 EOR
%   I:3.0/4  "Lug Loader Release PB" %
%   I:1.1/14  "Deck 1 Ducker downPB" %
%   B16:0/2  "Lug Loader Window" %
%   B16:0/6  "Lug Loader Manual feed" %
% Rung: 4 %
% Reset Manual Feed %
SOR XIO I:3.0/0 OSR B16:0/7 OTU B16:0/6 EOR
%   I:3.0/0  "Timber at Lug Loader Ducker" %
%   B16:0/6  "Lug Loader Manual feed" %
% Rung: 5 %
SOR XIO I:3.0/4 XIO I:1.1/14 OTU B16:0/6 EOR
%   I:3.0/4  "Lug Loader Release PB" %
%   I:1.1/14  "Deck 1 Ducker downPB" %
%   B16:0/6  "Lug Loader Manual feed" %

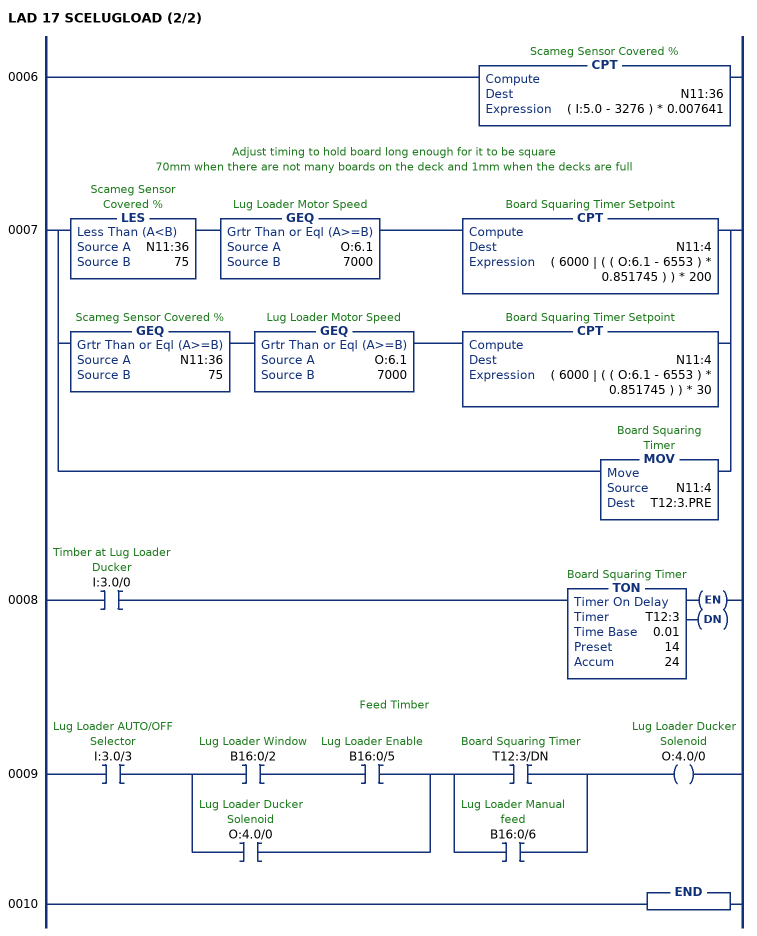
% Rung: 6 %
SOR CPT N11:36 " ( I:5.0 - 3276 ) * 0.007641 " EOR
%   N11:36  "Scameg Sensor Covered %" %
%   I:5.0  "Lug Loader Backlog %" %
% Rung: 7 %
% Adjust timing to hold board long enough for it to be square
%  70mm when there are not many boards on the deck and 1mm when the decks are full %
SOR BST LES N11:36 75 GEQ O:6.1 7000 CPT N11:4 " ( 6000 | ( ( O:6.1 - 6553 ) * 0.851745 ) ) * 200 " NXB GEQ N11:36 75 GEQ O:6.1 7000 CPT N11:4 " ( 6000 | ( ( O:6.1 - 6553 ) * 0.851745 ) ) * 30 " NXB MOV N11:4 T12:3.PRE BND EOR
%   N11:36  "Scameg Sensor Covered %" %
%   O:6.1  "Lug Loader Motor Speed" %
%   N11:4  "Board Squaring Timer Setpoint" %
%   T12:3  "Board Squaring Timer" %
% Rung: 8 %
SOR XIC I:3.0/0 TON T12:3 0.01 14 24 EOR
%   I:3.0/0  "Timber at Lug Loader Ducker" %
%   T12:3  "Board Squaring Timer" %
% Rung: 9 %
% Feed Timber %
SOR XIC I:3.0/3 BST XIC B16:0/2 XIC B16:0/5 NXB XIC O:4.0/0 BND BST XIC T12:3/DN NXB XIC B16:0/6 BND OTE O:4.0/0 EOR
%   I:3.0/3  "Lug Loader AUTO/OFF Selector" %
%   B16:0/2  "Lug Loader Window" %
%   B16:0/5  "Lug Loader Enable" %
%   O:4.0/0  "Lug Loader Ducker Solenoid" %
%   T12:3  "Board Squaring Timer" %
%   B16:0/6  "Lug Loader Manual feed" %
% Rung: 10 %
SOR END EOR

LADDER 18 "REPORTING"
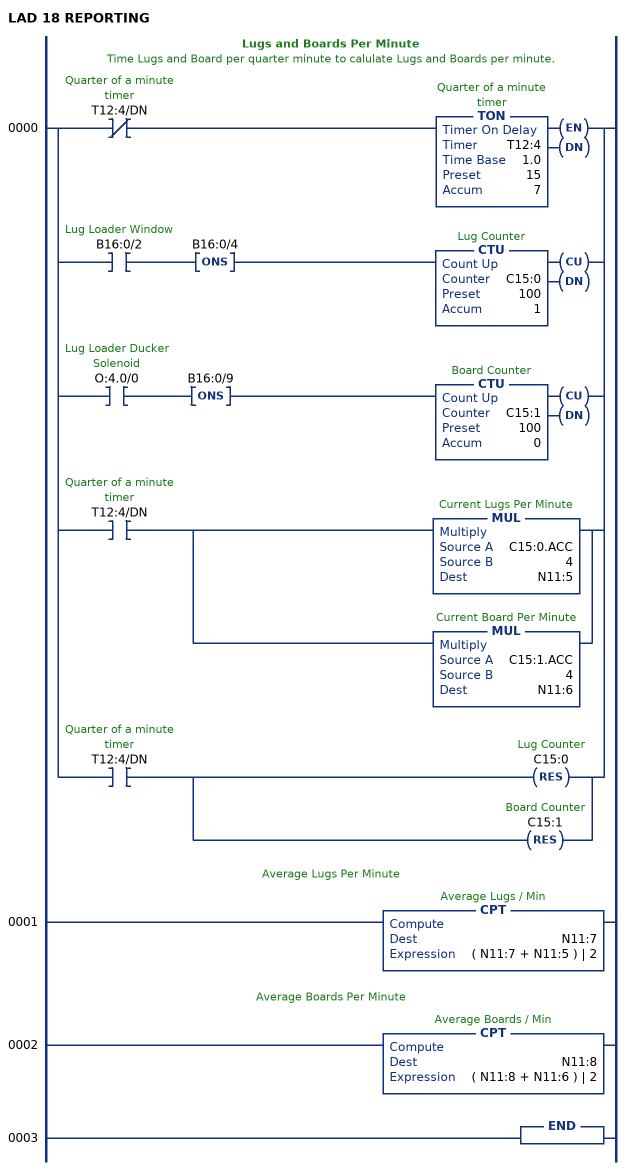
% Rung: 0 %
% TITLE: Lugs and Boards Per Minute %
% Time Lugs and Board per quarter minute to calulate Lugs and Boards per minute. %
SOR BST XIO T12:4/DN TON T12:4 1.0 15 7 NXB XIC B16:0/2 OSR B16:0/4 CTU C15:0 100 1 NXB XIC O:4.0/0 OSR B16:0/9 CTU C15:1 100 0 NXB XIC T12:4/DN BST MUL C15:0.ACC 4 N11:5 NXB MUL C15:1.ACC 4 N11:6 BND NXB XIC T12:4/DN BST RES C15:0 NXB RES C15:1 BND BND EOR
%   T12:4  "Quarter of a minute timer" %
%   B16:0/2  "Lug Loader Window" %
%   C15:0  "Lug Counter" %
%   O:4.0/0  "Lug Loader Ducker Solenoid" %
%   C15:1  "Board Counter" %
%   N11:5  "Current Lugs Per Minute" %
%   N11:6  "Current Board Per Minute" %
% Rung: 1 %
% Average Lugs Per Minute %
SOR CPT N11:7 " ( N11:7 + N11:5 ) | 2 " EOR
%   N11:7  "Average Lugs / Min" %
%   N11:5  "Current Lugs Per Minute" %
% Rung: 2 %
% Average Boards Per Minute %
SOR CPT N11:8 " ( N11:8 + N11:6 ) | 2 " EOR
%   N11:8  "Average Boards / Min" %
%   N11:6  "Current Board Per Minute" %
% Rung: 3 %
SOR END EOR

LADDER 20 "FILLET SYS"
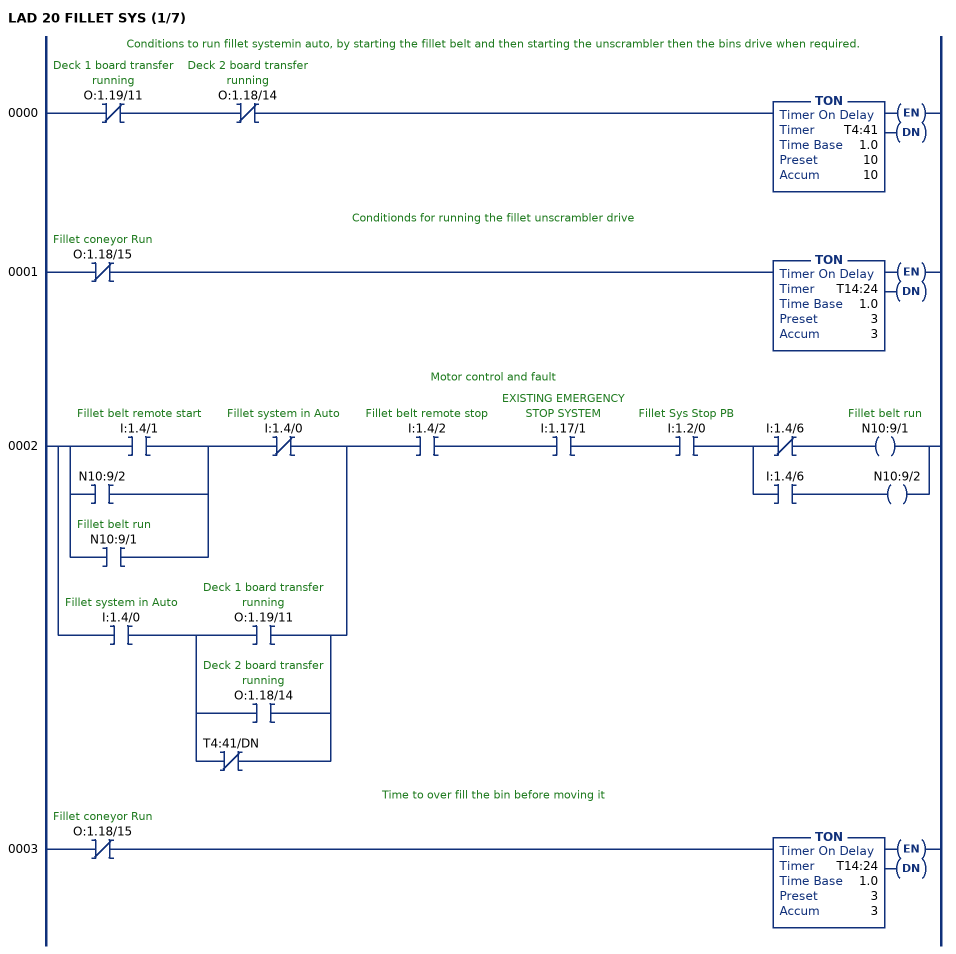
% Rung: 0 %
% Conditions to run fillet systemin auto, by starting the fillet belt and then starting the unscrambler then the bins drive when required. %
SOR XIO O:1.19/11 XIO O:1.18/14 TON T4:41 1.0 10 10 EOR
%   O:1.19/11  "Deck 1 board transfer running" %
%   O:1.18/14  "Deck 2 board transfer running" %
% Rung: 1 %
% Conditionds for running the fillet unscrambler drive %
SOR XIO O:1.18/15 TON T14:24 1.0 3 3 EOR
%   O:1.18/15  "Fillet coneyor Run" %
% Rung: 2 %
% Motor control and fault %
SOR BST BST XIC I:1.4/1 NXB XIC N10:9/2 NXB XIC N10:9/1 BND XIO I:1.4/0 NXB XIC I:1.4/0 BST XIC O:1.19/11 NXB XIC O:1.18/14 NXB XIO T4:41/DN BND BND XIC I:1.4/2 XIC I:1.17/1 XIC I:1.2/0 BST XIO I:1.4/6 OTE N10:9/1 NXB XIC I:1.4/6 OTE N10:9/2 BND EOR
%   I:1.4/1  "Fillet belt remote start" %
%   N10:9/1  "Fillet belt run" %
%   I:1.4/0  "Fillet system in Auto" %
%   O:1.19/11  "Deck 1 board transfer running" %
%   O:1.18/14  "Deck 2 board transfer running" %
%   I:1.4/2  "Fillet belt remote stop" %
%   I:1.17/1  "EXISTING EMERGENCY STOP SYSTEM" %
%   I:1.2/0  "Fillet Sys Stop PB" %
% Rung: 3 %
% Time to over fill the bin before moving it %
SOR XIO O:1.18/15 TON T14:24 1.0 3 3 EOR
%   O:1.18/15  "Fillet coneyor Run" %

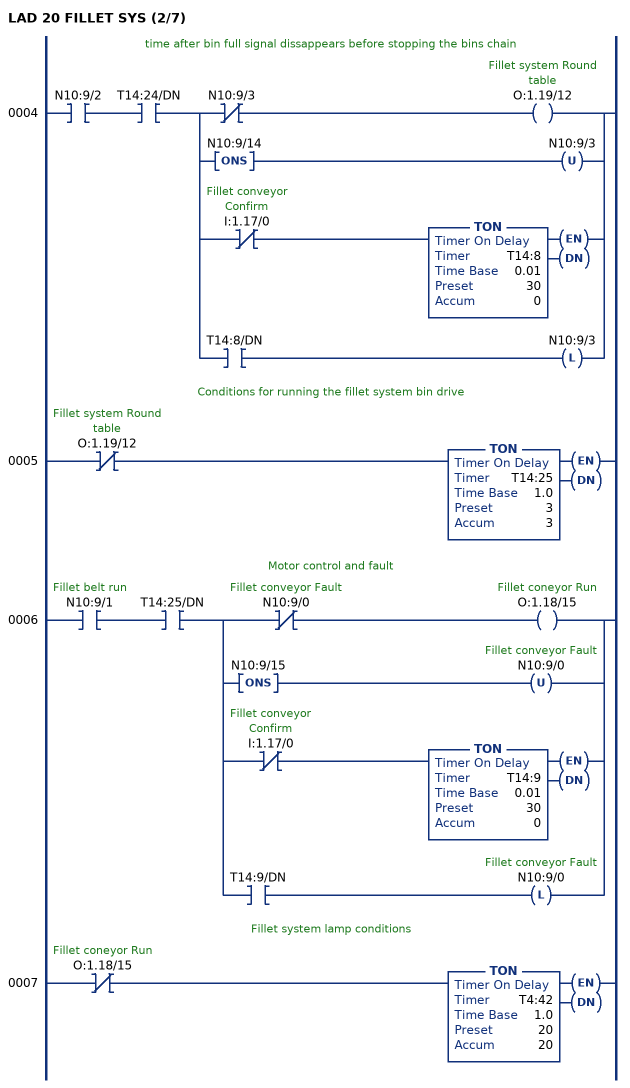
% Rung: 4 %
% time after bin full signal dissappears before stopping the bins chain %
SOR XIC N10:9/2 XIC T14:24/DN BST XIO N10:9/3 OTE O:1.19/12 NXB OSR N10:9/14 OTU N10:9/3 NXB XIO I:1.17/0 TON T14:8 0.01 30 0 NXB XIC T14:8/DN OTL N10:9/3 BND EOR
%   O:1.19/12  "Fillet system Round table" %
%   I:1.17/0  "Fillet conveyor Confirm" %
% Rung: 5 %
% Conditions for running the fillet system bin drive %
SOR XIO O:1.19/12 TON T14:25 1.0 3 3 EOR
%   O:1.19/12  "Fillet system Round table" %
% Rung: 6 %
% Motor control and fault %
SOR XIC N10:9/1 XIC T14:25/DN BST XIO N10:9/0 OTE O:1.18/15 NXB OSR N10:9/15 OTU N10:9/0 NXB XIO I:1.17/0 TON T14:9 0.01 30 0 NXB XIC T14:9/DN OTL N10:9/0 BND EOR
%   N10:9/1  "Fillet belt run" %
%   N10:9/0  "Fillet conveyor Fault" %
%   O:1.18/15  "Fillet coneyor Run" %
%   I:1.17/0  "Fillet conveyor Confirm" %
% Rung: 7 %
% Fillet system lamp conditions %
SOR XIO O:1.18/15 TON T4:42 1.0 20 20 EOR
%   O:1.18/15  "Fillet coneyor Run" %

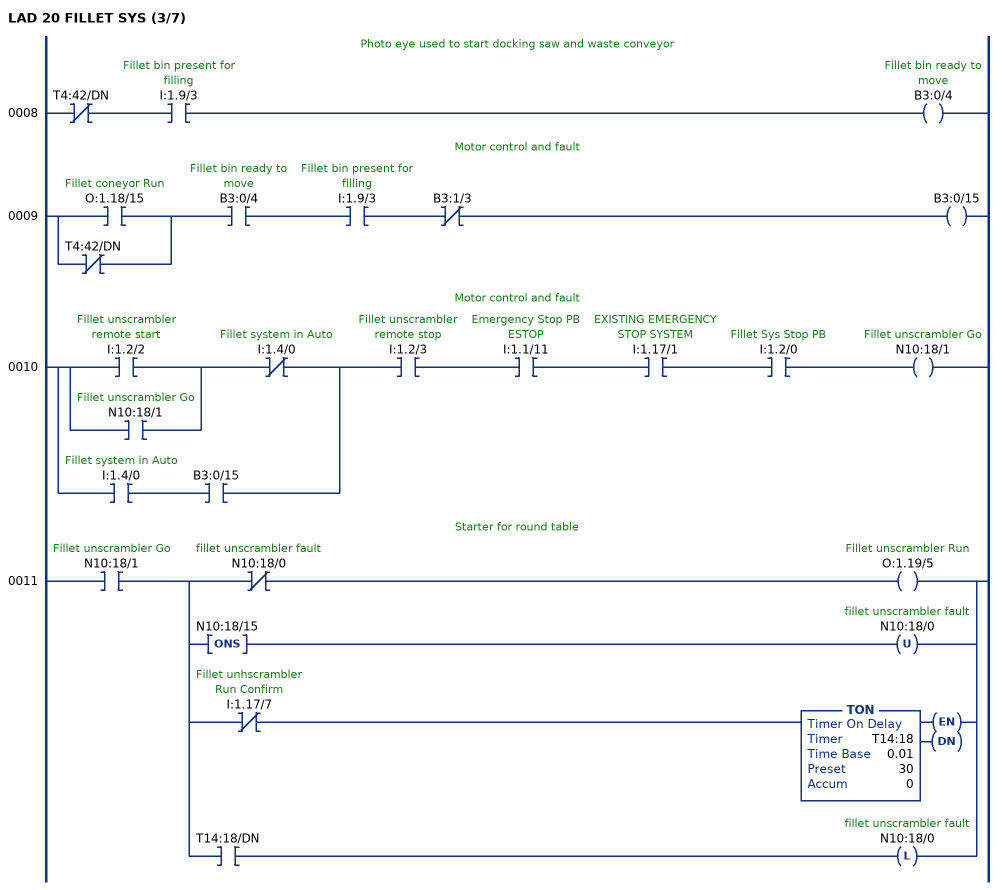
% Rung: 8 %
% Photo eye used to start docking saw and waste conveyor %
SOR XIO T4:42/DN XIC I:1.9/3 OTE B3:0/4 EOR
%   I:1.9/3  "Fillet bin present for filling" %
%   B3:0/4  "Fillet bin ready to move" %
% Rung: 9 %
% Motor control and fault %
SOR BST XIC O:1.18/15 NXB XIO T4:42/DN BND XIC B3:0/4 XIC I:1.9/3 XIO B3:1/3 OTE B3:0/15 EOR
%   O:1.18/15  "Fillet coneyor Run" %
%   B3:0/4  "Fillet bin ready to move" %
%   I:1.9/3  "Fillet bin present for filling" %
% Rung: 10 %
% Motor control and fault %
SOR BST BST XIC I:1.2/2 NXB XIC N10:18/1 BND XIO I:1.4/0 NXB XIC I:1.4/0 XIC B3:0/15 BND XIC I:1.2/3 XIC I:1.1/11 XIC I:1.17/1 XIC I:1.2/0 OTE N10:18/1 EOR
%   I:1.2/2  "Fillet unscrambler remote start" %
%   N10:18/1  "Fillet unscrambler Go" %
%   I:1.4/0  "Fillet system in Auto" %
%   I:1.2/3  "Fillet unscrambler remote stop" %
%   I:1.1/11  ESTOP  "Emergency Stop PB" %
%   I:1.17/1  "EXISTING EMERGENCY STOP SYSTEM" %
%   I:1.2/0  "Fillet Sys Stop PB" %
% Rung: 11 %
% Starter for round table %
SOR XIC N10:18/1 BST XIO N10:18/0 OTE O:1.19/5 NXB OSR N10:18/15 OTU N10:18/0 NXB XIO I:1.17/7 TON T14:18 0.01 30 0 NXB XIC T14:18/DN OTL N10:18/0 BND EOR
%   N10:18/1  "Fillet unscrambler Go" %
%   N10:18/0  "fillet unscrambler fault" %
%   O:1.19/5  "Fillet unscrambler Run" %
%   I:1.17/7  "Fillet unhscrambler Run Confirm" %

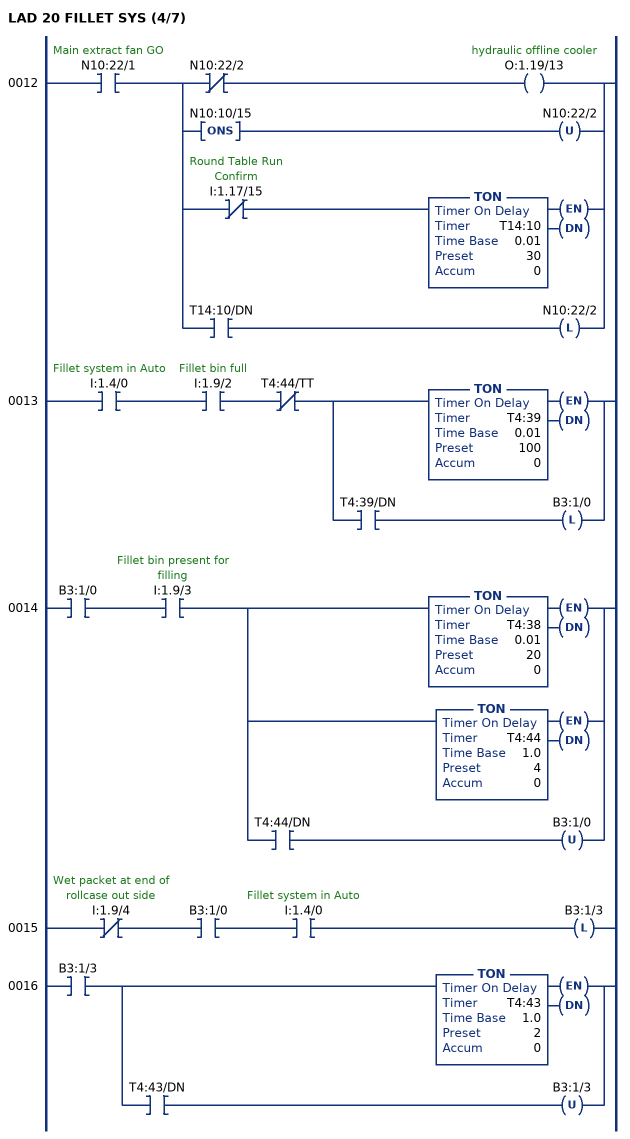
% Rung: 12 %
SOR XIC N10:22/1 BST XIO N10:22/2 OTE O:1.19/13 NXB OSR N10:10/15 OTU N10:22/2 NXB XIO I:1.17/15 TON T14:10 0.01 30 0 NXB XIC T14:10/DN OTL N10:22/2 BND EOR
%   N10:22/1  "Main extract fan GO" %
%   O:1.19/13  "hydraulic offline cooler" %
%   I:1.17/15  "Round Table Run Confirm" %
% Rung: 13 %
SOR XIC I:1.4/0 XIC I:1.9/2 XIO T4:44/TT BST TON T4:39 0.01 100 0 NXB XIC T4:39/DN OTL B3:1/0 BND EOR
%   I:1.4/0  "Fillet system in Auto" %
%   I:1.9/2  "Fillet bin full" %
% Rung: 14 %
SOR XIC B3:1/0 XIC I:1.9/3 BST TON T4:38 0.01 20 0 NXB TON T4:44 1.0 4 0 NXB XIC T4:44/DN OTU B3:1/0 BND EOR
%   I:1.9/3  "Fillet bin present for filling" %
% Rung: 15 %
SOR XIO I:1.9/4 XIC B3:1/0 XIC I:1.4/0 OTL B3:1/3 EOR
%   I:1.9/4  "Wet packet at end of rollcase out side" %
%   I:1.4/0  "Fillet system in Auto" %
% Rung: 16 %
SOR XIC B3:1/3 BST TON T4:43 1.0 2 0 NXB XIC T4:43/DN OTU B3:1/3 BND EOR

